FUNCTION F_LRealToStringEx : STRING(255)
VAR_INPUT
	fValue: LREAL;
	iPrecision: INT := 3;
END_VAR
VAR
	fbFormat: FB_FormatString;
END_VAR

fbFormat( sFormat := Concat3('%.', INT_TO_STRING(iPrecision), 'f'), arg1 := F_LREAL( fValue ), sOut => F_LRealToStringEx);

END_FUNCTION

(* stored: Version 1.1.0.1, ProductVersion 3.1.4022.9
   POU F_LRealToStringEx: Id {5ad64110-40a8-4271-8a35-abc9d6257b76}, SpecialFunc None *)
